FUNCTION_BLOCK FB_Actuator IMPLEMENTS IActuator
VAR_INPUT
END_VAR
VAR_OUTPUT
END_VAR
VAR
	bExtended			AT %I* : BOOL;
	bRetracted			AT %I* : BOOL;
	bExtendCmd			AT %Q* : BOOL;
	bRetractCmd			AT %Q* : BOOL;
	
	iCycleState			: DINT;
	bError				: BOOL;
	tmrTimeout			: TON;
END_VAR

METHOD Cycle : BOOL
CASE iCycleState OF
	0:
		IF Extend() THEN
			iCycleState := 1;
		END_IF
	1:
		IF Retract() THEN
			iCycleState := 2;
		END_IF
		
	2:
		iCycleState := 0;
		Cycle := TRUE;
END_CASE
END_METHOD

PROPERTY Error : BOOL
GET
Error := bError;
END_GET
END_PROPERTY

METHOD Extend : BOOL
bRetractCmd := FALSE;
bExtendCmd := TRUE;
IF bExtended THEN
	bExtendCmd := FALSE;
	bError := FALSE;
	tmrTimeout(IN:=FALSE);
	Extend := TRUE;
ELSE
	tmrTimeout(IN:=TRUE, PT:=T#5S);
	IF tmrTimeout.Q THEN
		bError := TRUE;
	END_IF
END_IF
END_METHOD

PROPERTY Extended : BOOL
GET
Extended := bExtended;
END_GET
END_PROPERTY

METHOD Retract : BOOL
bExtendCmd := FALSE;
bRetractCmd := TRUE;
IF bRetracted THEN
	bRetractCmd := FALSE;
	bError := FALSE;
	tmrTimeout(IN:=FALSE);
	Retract := TRUE;
ELSE
	tmrTimeout(IN:=TRUE, PT:=T#5S);
	IF tmrTimeout.Q THEN
		bError := TRUE;
	END_IF
END_IF
END_METHOD

PROPERTY Retracted : BOOL
GET
Retracted := bRetracted;
END_GET
END_PROPERTY

END_FUNCTION_BLOCK

(* stored: Version 1.1.0.1, ProductVersion 3.1.4024.12
   POU FB_Actuator: Id {b60feaab-d854-40dc-b58d-c92ca4bd5a91}, SpecialFunc None
   Method Cycle: Id {37965100-d96c-4645-8c71-ca1df0408b13}
   Property Error: Id {9ba52509-1d4d-4275-9de2-387c1d3da456}
   Get Get: Id {ad289723-a406-4fec-92f9-b69f75d3f237}
   Method Extend: Id {40a95e29-a632-41af-a987-4c935a3fa911}
   Property Extended: Id {b8ac5087-3ff2-43a7-b584-1f32518f4381}
   Get Get: Id {adb61051-46e0-4181-8afd-273eaf7161cb}
   Method Retract: Id {55bc305c-9eba-4946-bab0-3b5fb897cca8}
   Property Retracted: Id {9945b710-2862-4e2a-92dd-863f037f83ee}
   Get Get: Id {52d1f740-9588-4293-91ea-6e94a1c38ca8} *)
